TYPE libT_Char : STRING[1];
END_TYPE

(* stored: Version 1.1.0.1
   DUT libT_Char: Id {7c71d900-3c68-401d-92e1-3340e4c158e6} *)
